FUNCTION_BLOCK FB_FlyPowerMarkExeManager
VAR_INPUT
	UpsPowerStatus : E_UpsPowerStatus;
	LasitControllerOn : BOOL;
	Reset : BOOL;
END_VAR
VAR_OUTPUT
	Error	: BOOL  := FALSE;
	ErrorID	: INT 	:= 0;
	ErrorSubID	: INT 	:= 0;
END_VAR
VAR_IN_OUT
	Init	: BOOL;
	NT_OpenExe : NT_StartProcess;
	NT_CloseExe : NT_StartProcess;
END_VAR
VAR
	iState				: INT 	:= 0;
	RTRIG_PowerOnLine	: R_TRIG;
	RTRIG_PowerOnBattery	: R_TRIG;
	RTRIG_Reset			: R_TRIG;
	DelayOpenExe		: TON;
	TON_Timeout			: TON;
	tTimeout			: TIME := T#10S;
END_VAR

RTRIG_PowerOnLine(CLK := UpsPowerStatus = E_UpsPowerStatus.PowerOnLine);
RTRIG_PowerOnBattery(CLK := UpsPowerStatus = E_UpsPowerStatus.PowerOnBattery);

RTRIG_Reset(CLK := Reset);
IF RTRIG_Reset.Q THEN
	iState := 0;
	ErrorID 	:= 0;
	ErrorSubID := 0;
	Error		:= FALSE;
END_IF

IF RTRIG_PowerOnLine.Q THEN
	NT_OpenExe.START := FALSE;
	NT_CloseExe.START := FALSE;
	iState := 10;
END_IF

IF RTRIG_PowerOnBattery.Q THEN
	NT_OpenExe.START := FALSE;
	NT_CloseExe.START := FALSE;
	iState := 100;
END_IF

DelayOpenExe(IN := iState = 10 AND LasitControllerOn, PT := T#30S);

CASE iState OF
	0:
		;
		
	10:
		IF Init THEN
			Init := FALSE;
			iState := 0;
		ELSIF DelayOpenExe.Q THEN
			//NT_OpenExe.COMNDLINE := 'FLY_POWERMARK.exe "C:\Program Files (x86)\Lasit spa\Laser_FLY_POWERMARK\FLY_POWERMARK.exe"'; 
			//togliere commento se si vuole attivare debug dell'esecuzione del .bat
			NT_OpenExe.COMNDLINE := 'FLY_POWERMARK.exe "C:\Program Files (x86)\Lasit spa\Laser_FLY_POWERMARK\FLY_POWERMARK.exe" debug'; 
		
			iState := 20;
		END_IF
		
	20:
		NT_OpenExe.START := TRUE;
		IF NT_OpenExe.BUSY THEN
			iState := 30;
		END_IF
		
	30:
		IF NOT NT_OpenExe.BUSY THEN
			NT_OpenExe.START := FALSE;
			iState := 0;
		ELSIF NT_OpenExe.ERR THEN
			NT_OpenExe.START := FALSE;
			iStateError();
		END_IF		

	100:
		//NT_CloseExe.COMNDLINE := 'FLY_POWERMARK.exe';
		//togliere commento se si vuole attivare debug dell'esecuzione del .bat
		NT_CloseExe.COMNDLINE := 'FLY_POWERMARK.exe debug';
		iState := 110;
		
	110:
		NT_CloseExe.START := TRUE;
		IF NT_CloseExe.BUSY THEN
			iState := 120;
		END_IF
		
	120:
		IF NOT NT_CloseExe.BUSY THEN
			NT_CloseExe.START := FALSE;
			iState := 0;
		ELSIF NT_CloseExe.ERR THEN
			NT_CloseExe.START := FALSE;
			iStateError();
		END_IF		
	
END_CASE

//Timeout
Timeout();

// ERROR
ErrorSet();

METHOD PRIVATE ErrorSet : BOOL
IF (iState >= 1000) THEN
	ErrorID 	:= iState;
	Error		:= TRUE;
	ErrorSet	:= TRUE;
	
	iState		:= -1;
ELSE
	ErrorSet := FALSE;
END_IF
END_METHOD

METHOD PRIVATE iStateError
iState := iState + 1000;
END_METHOD

METHOD PRIVATE Timeout : BOOL
TON_Timeout(IN:= iState > 0 AND iState < 1000 AND iState <> 10 AND tTimeout <> T#0MS, PT := tTimeout);
IF TON_Timeout.Q THEN
    ErrorSubID := iState;
	Timeout := TRUE;
	
    iState := 1999;
ELSE
	Timeout := FALSE;
END_IF
END_METHOD

END_FUNCTION_BLOCK

(* stored: Version 1.1.0.1, ProductVersion 3.1.4024.15
   POU FB_FlyPowerMarkExeManager: Id {19f9f03b-3f88-410a-8010-1b63f38f8a87}, SpecialFunc None
   Method ErrorSet: Id {199bfb96-eba9-4e9a-b0b2-64f1de3fa7ef}
   Method iStateError: Id {c9c18385-2936-4bff-bdad-4aa8e3dfbf86}
   Method Timeout: Id {96760c1b-b35a-4484-a00d-3cecb4d146bc} *)
